INTERFACE I_Observer EXTENDS __System.IQueryInterface

METHOD Update : BYTE
VAR_INPUT
	nNewValue		: BYTE(0..100);
END_VAR
END_METHOD

END_INTERFACE

(* stored: Version 1.1.0.1, ProductVersion 3.1.4024.9
   Itf I_Observer: Id {ad922435-6e6d-45d3-94ba-ef34a18789aa}
   Method Update: Id {975a63c2-7d49-4b17-9936-5f690435e016} *)
